SUBAPPLICATION StringValue_TO_NVS (* String-VT-Wert einlesen und in NVS speichern (generisch). *)
  (* Standard: 61499-2 *)
  (* Version 1.0, 2026-09-09, Franz Höpfinger, Meisterschulen am Ostbahnhof, Ausgelagert aus Uebung_012m_sub zur Wiederverwendung. *)
  PACKAGE MyLib::sys;
  IMPORT isobus::UT::Q::const::IDs::ID_NULL;
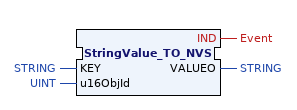
  EVENT_OUTPUT
    IND;
  END_EVENT
  VAR_INPUT
    KEY : STRING; (* Key name. *)
    u16ObjId : UINT := ID_NULL;
  END_VAR
  VAR_OUTPUT
    VALUEO : STRING;
  END_VAR
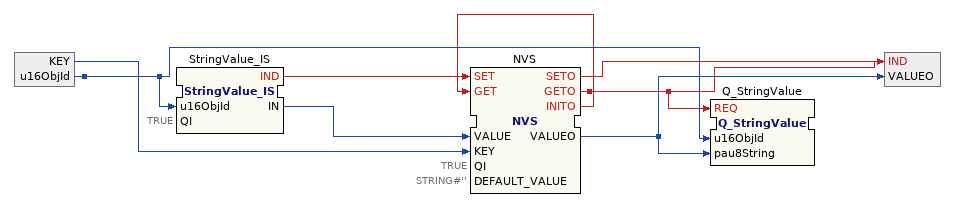
  FBS
    StringValue_IS : isobus::UT::io::StringValue::StringValue_IS(QI := TRUE);
    NVS : logiBUS::storage::esp32_nvs::NVS(QI := TRUE, DEFAULT_VALUE := STRING#'');
    Q_StringValue : isobus::UT::Q::Q_StringValue;
  END_FBS
  EVENT_CONNECTIONS
    StringValue_IS.IND TO NVS.SET;
    NVS.SETO TO IND;
    NVS.GETO TO Q_StringValue.REQ;
    NVS.GETO TO IND;
    NVS.INITO TO NVS.GET;
  END_CONNECTIONS
  DATA_CONNECTIONS
    StringValue_IS.IN TO NVS.VALUE;
    u16ObjId TO Q_StringValue.u16ObjId;
    KEY TO NVS.KEY;
    NVS.VALUEO TO Q_StringValue.pau8String;
    NVS.VALUEO TO VALUEO;
    u16ObjId TO StringValue_IS.u16ObjId;
  END_CONNECTIONS
END_SUBAPPLICATION
